// TIA Portal V18 export
FUNCTION_BLOCK "FB10-heater"   // FB12, LAD
{ S7_Optimized_Access := 'TRUE' }
VERSION : 0.1
// stored: AutoNumber true, IsIECCheckEnabled false, IsRetainMemResEnabled false, MemoryReserve 100, SetENOAutomatically false, UDAEnableTagReadback false
   VAR_INPUT
      ON : Bool;
      "Temperature oC" : Real;
      "Set temperature" : Real;
      "pre shutdown temperature" : Real;
      "Limit under temperature" : Real;
      "Limit Over temperature" : Real;
      "heating adjustment hysteresis" : Real;
      "Minimum ON time" : Real;
      "Minimum OFF time" : Real;
   END_VAR
   VAR_OUTPUT
      "Heater PWM" : Bool;
      "Heater Temperature under Limit" : Bool;
      "Heater Temperature Over Limit" : Bool;
      "Temperature Above SP" { ExternalAccessible := 'False'; ExternalVisible := 'False'; ExternalWritable := 'False'} : Bool;
      "Dispensing Stop undertemperature" { ExternalAccessible := 'False'; ExternalVisible := 'False'; ExternalWritable := 'False'} : Bool;
   END_VAR
   VAR
      "set temperature after hysteresis" : Real;
      "On time in msec" : DInt;
      "off time in msec" : DInt;
      "On timer triggered" : Bool;
      "off time triggered" : Bool;
      IEC_Timer_0_Instance { S7_SetPoint := 'True'} : TON_TIME;
      IEC_Timer_0_Instance_1 { S7_SetPoint := 'True'} : TON_TIME;
   END_VAR
   VAR_TEMP   // added for the SCL form of the ladder/FBD networks
      _w1 : Bool;
   END_VAR
BEGIN

REGION Network 1: On/off timer in sec
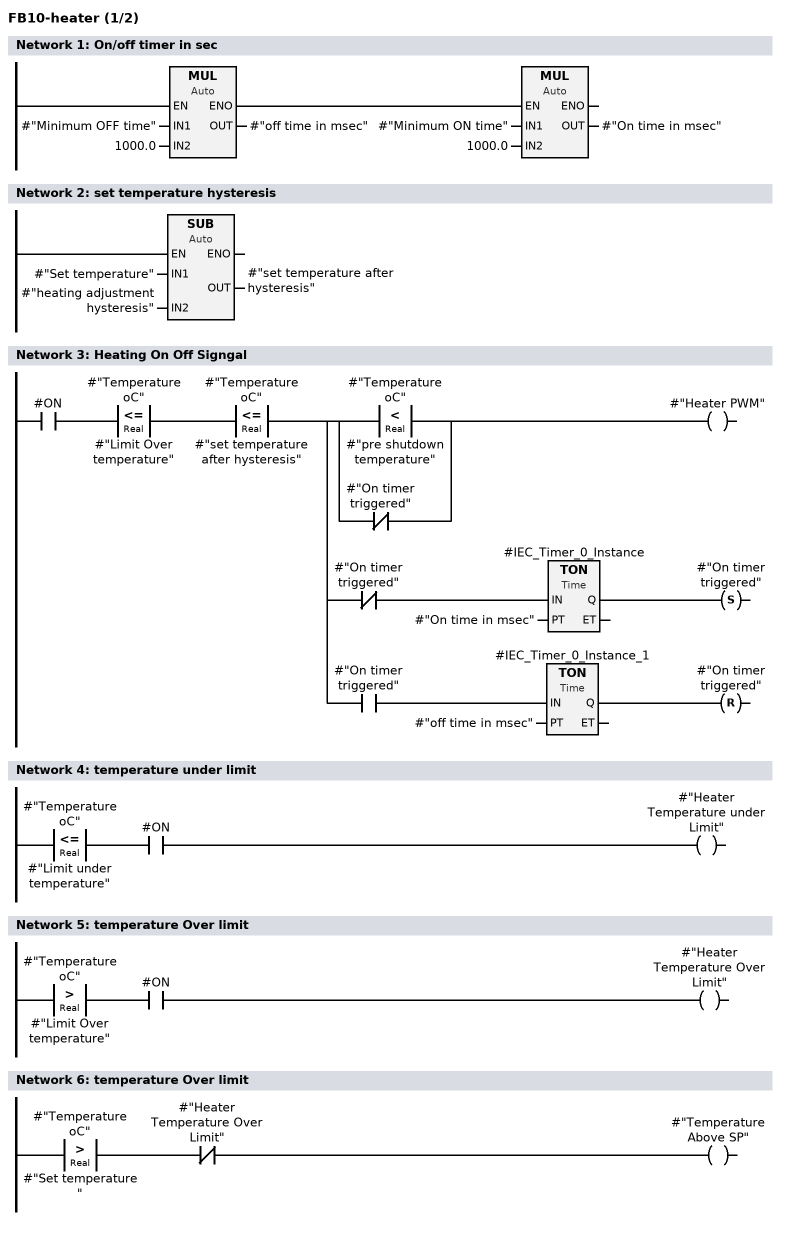
   RUNG wire#powerrail
      Mul(in1 := #"Minimum OFF time", in2 := 1000.0, out => #"off time in msec")
      Mul(in1 := #"Minimum ON time", in2 := 1000.0, out => #"On time in msec")
   END_RUNG
   // the same network as SCL:
   #"off time in msec" := #"Minimum OFF time" * 1000.0;
   #"On time in msec" := #"Minimum ON time" * 1000.0;
END_REGION

REGION Network 2: set temperature hysteresis
   RUNG wire#powerrail
      Sub(in1 := #"Set temperature", in2 := #"heating adjustment hysteresis", out => #"set temperature after hysteresis")
   END_RUNG
   // the same network as SCL:
   #"set temperature after hysteresis" := #"Set temperature" - #"heating adjustment hysteresis";
END_REGION

REGION Network 3: Heating On Off Signgal
   RUNG wire#powerrail
      Contact( #ON )
      { S7_Templates := "SrcType := Real" } LE_Contact(in1 := #"Temperature oC", in2 := #"Limit Over temperature")
      { S7_Templates := "SrcType := Real" } LE_Contact(in1 := #"Temperature oC", in2 := #"set temperature after hysteresis")
      wire#w1
      { S7_Templates := "SrcType := Real" } LT_Contact(in1 := #"Temperature oC", in2 := #"pre shutdown temperature")
      wire#w2
      Coil( #"Heater PWM" )
   END_RUNG
   RUNG wire#w1
      I_Contact( #"On timer triggered" )
   END_RUNG wire#w2
   RUNG wire#w1
      I_Contact( #"On timer triggered" )
      { S7_Templates := "time_type := Time" } #IEC_Timer_0_Instance.TON(pt := #"On time in msec", et =>)
      S_Coil( #"On timer triggered" )
   END_RUNG
   RUNG wire#w1
      Contact( #"On timer triggered" )
      { S7_Templates := "time_type := Time" } #IEC_Timer_0_Instance_1.TON(pt := #"off time in msec", et =>)
      R_Coil( #"On timer triggered" )
   END_RUNG
   // the same network as SCL:
   #_w1 := #ON AND (#"Temperature oC" <= #"Limit Over temperature") AND (#"Temperature oC" <= #"set temperature after hysteresis");
   #"Heater PWM" := #_w1 AND ((#"Temperature oC" < #"pre shutdown temperature") OR NOT #"On timer triggered");
   #IEC_Timer_0_Instance(IN := #_w1 AND NOT #"On timer triggered", PT := #"On time in msec");   // TON
   IF #IEC_Timer_0_Instance.Q THEN #"On timer triggered" := TRUE; END_IF;
   #IEC_Timer_0_Instance_1(IN := #_w1 AND #"On timer triggered", PT := #"off time in msec");   // TON
   IF #IEC_Timer_0_Instance_1.Q THEN #"On timer triggered" := FALSE; END_IF;
END_REGION

REGION Network 4: temperature under limit
   RUNG wire#powerrail
      { S7_Templates := "SrcType := Real" } LE_Contact(in1 := #"Temperature oC", in2 := #"Limit under temperature")
      Contact( #ON )
      Coil( #"Heater Temperature under Limit" )
   END_RUNG
   // the same network as SCL:
   #"Heater Temperature under Limit" := (#"Temperature oC" <= #"Limit under temperature") AND #ON;
END_REGION

REGION Network 5: temperature Over limit
   RUNG wire#powerrail
      { S7_Templates := "SrcType := Real" } GT_Contact(in1 := #"Temperature oC", in2 := #"Limit Over temperature")
      Contact( #ON )
      Coil( #"Heater Temperature Over Limit" )
   END_RUNG
   // the same network as SCL:
   #"Heater Temperature Over Limit" := (#"Temperature oC" > #"Limit Over temperature") AND #ON;
END_REGION

REGION Network 6: temperature Over limit
   RUNG wire#powerrail
      { S7_Templates := "SrcType := Real" } GT_Contact(in1 := #"Temperature oC", in2 := #"Set temperature")
      I_Contact( #"Heater Temperature Over Limit" )
      Coil( #"Temperature Above SP" )
   END_RUNG
   // the same network as SCL:
   #"Temperature Above SP" := (#"Temperature oC" > #"Set temperature") AND NOT #"Heater Temperature Over Limit";
END_REGION

REGION Network 7: Temperature Under limit to Stop Dispensing
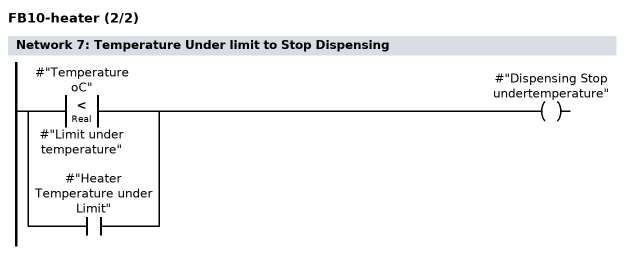
   RUNG wire#powerrail
      { S7_Templates := "SrcType := Real" } LT_Contact(in1 := #"Temperature oC", in2 := #"Limit under temperature")
      wire#w1
      Coil( #"Dispensing Stop undertemperature" )
   END_RUNG
   RUNG wire#powerrail
      Contact( #"Heater Temperature under Limit" )
   END_RUNG wire#w1
   // the same network as SCL:
   #"Dispensing Stop undertemperature" := (#"Temperature oC" < #"Limit under temperature") OR #"Heater Temperature under Limit";
END_REGION
END_FUNCTION_BLOCK
